PROGRAM MAIN
VAR
	_fb : FB_ST10; 
END_VAR

_fb._scanner();

END_PROGRAM

(* stored: Version 1.1.0.1, ProductVersion 3.1.4024.12
   POU MAIN: Id {5a8e1327-26d3-4e43-8559-97c135f86653}, SpecialFunc None *)
